TYPE ToolDataX :
STRUCT
	{attribute 'OPC.UA.DA.Description' := 'Unique ID of Tool'}
	TooID					: UINT;

	{attribute 'OPC.UA.DA.Description' := 'ID of the location of Tool'}
	Location				: UINT;

	{attribute 'OPC.UA.DA.Description' := 'Usage cycles since tool configuration'}
	CurrentCycles			: UDINT;

	{attribute 'OPC.UA.DA.Description' := 'Max allowed cycles for tool'}
	MaxCycles				: UDINT;

END_STRUCT
END_TYPE

(* stored: Version 1.1.0.1, ProductVersion 3.1.4024.5
   DUT ToolDataX: Id {679837d4-dbba-4451-896c-221972c607dd} *)
